{attribute 'qualified_only'}
VAR_GLOBAL CONSTANT
	cServiceCount : UINT := SIZEOF(ST_GC_ServiceCtrl) / SIZEOF(ST_PML_Base_In);
END_VAR

(* stored: Version 1.1.0.1, ProductVersion 3.1.4026.18
   GVL GVL_GC_Config: Id {e17c4bd1-c3da-471b-9592-c1512b9dedb8} *)
